FUNCTION_BLOCK a3 (* Basic FB with empty ECC *)
  (* Standard: 61499-2 *)
  (* Version 1.0, 2025-03-31, 06220625900 *)
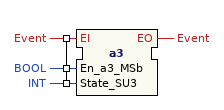
  EVENT_INPUT
    EI WITH En_a3_MSb, State_SU3;
  END_EVENT
  EVENT_OUTPUT
    EO;
  END_EVENT
  VAR_INPUT
    En_a3_MSb : BOOL := False;
    State_SU3 : INT := 1;
  END_VAR
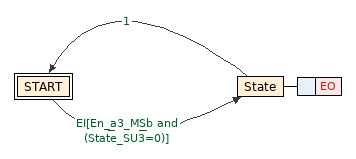
  EC_STATES
    START; (* Initial State *)
    State : -> EO;
  END_STATES
  EC_TRANSITIONS
    START TO State := EI[En_a3_MSb and (State_SU3=0)];
    State TO START := 1;
  END_TRANSITIONS
END_FUNCTION_BLOCK
